// TIA Portal V17 export
// export: Created 2023-03-08T06:46:29.0432064Z, ExportSetting WithDefaults, DisplayName Totally Integrated Automation Portal, DisplayVersion V17 Update 4, DisplayName TIA Portal Openness, DisplayVersion V17 Update 4, DisplayName TIA Portal Version Control Interface, DisplayVersion V17, DisplayName STEP 7 Professional, DisplayVersion V17 Update 4, DisplayName STEP 7 Safety, DisplayVersion V17, DisplayName WinCC Professional, DisplayVersion V17 Update 4
DATA_BLOCK "EME"   // DB502, F_DB
{ S7_Optimized_Access := 'TRUE' }
VERSION : 0.1
// stored: AutoNumber false, DBAccessibleFromOPCUA true, DBAccessibleFromWebserver true
   VAR
      xAlwaysOff : Bool;
      xBattOpenCmd : Bool;
      xStopPCSCmd : Bool;
      xMVbrkOpenCmd : Bool;
      xMVtrafoSt : Bool;
      xAuxSkid : Bool;
      xAuxSkidDelay : Bool;
      xAuxSkidFireMan : Bool;
      xAuxSkidFireManDelay : Bool;
      xCore : Bool;
      xCoreDelay : Bool;
      xTwinPCS : Bool;
      xPCSCmd : Bool;
      xResetCmd : Bool;
      xByPass : Bool;
      xRcvError : Bool;
      xSendError : Bool;
      xAckReq : Bool;
      xByPassCore : Bool;
   END_VAR
BEGIN
END_DATA_BLOCK
